{attribute addProperty BoxType "EP2328-1061-0016"}
{attribute addProperty Id "DI_X01_Pin4_InputAT %I*DI_X01_Pin4_Input_E4AEF59E810DI_X01_Pin2_InputAT %I*DI_X01_Pin2_Input_E4AEF59E810DI_X02_Pin4_InputAT %I*DI_X02_Pin4_Input_E4AEF59E810DI_X02_Pin2_InputAT %I*DI_X02_Pin2_Input_E4AEF59E810DO_X03_Pin4_OutputAT %Q*DO_X03_Pin4_Output_7F374EB0810DO_X03_Pin2_OutputAT %Q*DO_X03_Pin2_Output_7F374EB0810DO_X04_Pin4_OutputAT %Q*DO_X04_Pin4_Output_7F374EB0810DO_X04_Pin2_OutputAT %Q*DO_X04_Pin2_Output_7F374EB0810WcStateAT %I*WcState_98A4DF7520.250InfoDataAT %I*InfoData_192954DE1620"}
{attribute addProperty CRC "965961157"}
{attribute addProperty SizeInBites "82"}
{attribute addProperty SizeInBytes "10.25"}
TYPE EP2328_FBC9733E :
STRUCT
	{attribute addProperty Name "DI_X01_Pin4_Input"}
	DI_X01_Pin4_Input : DI_X01_Pin4_Input_E4AEF59E;
	{attribute addProperty Name "DI_X01_Pin2_Input"}
	DI_X01_Pin2_Input : DI_X01_Pin2_Input_E4AEF59E;
	{attribute addProperty Name "DI_X02_Pin4_Input"}
	DI_X02_Pin4_Input : DI_X02_Pin4_Input_E4AEF59E;
	{attribute addProperty Name "DI_X02_Pin2_Input"}
	DI_X02_Pin2_Input : DI_X02_Pin2_Input_E4AEF59E;
	{attribute addProperty Name "DO_X03_Pin4_Output"}
	DO_X03_Pin4_Output : DO_X03_Pin4_Output_7F374EB0;
	{attribute addProperty Name "DO_X03_Pin2_Output"}
	DO_X03_Pin2_Output : DO_X03_Pin2_Output_7F374EB0;
	{attribute addProperty Name "DO_X04_Pin4_Output"}
	DO_X04_Pin4_Output : DO_X04_Pin4_Output_7F374EB0;
	{attribute addProperty Name "DO_X04_Pin2_Output"}
	DO_X04_Pin2_Output : DO_X04_Pin2_Output_7F374EB0;
	{attribute addProperty Name "WcState"}
	WcState : WcState_98A4DF75;
	{attribute addProperty Name "InfoData"}
	InfoData : InfoData_192954DE;
END_STRUCT
END_TYPE

(* stored: Version 1.2.0.0, ProductVersion 3.1.4024.9
   DUT EP2328_FBC9733E: Id {63605aa1-78eb-4510-9a79-677d0cb7efe8} *)
